(* Logix 5000 project; controller Test Emulate 5570 rev 32.11; software revision 32.00 *)

TASK MainTask (continuous, watchdog 500 ms) : MainProgram

MODULES
   Local : Emulate 5570 (ICP 5, rev 32.11)
END_MODULES

TYPE Jeyc_data :
STRUCT
   a : BOOL;
   b : BOOL;
   c : BOOL;
END_STRUCT
END_TYPE

TYPE TestUDT :
STRUCT
   b : BOOL;
END_STRUCT
END_TYPE

VAR_GLOBAL   (* controller tags *)
   HOLD : BOOL; {access Read Only}
   PROG1 : BOOL; {access Read Only}
   PROG2 : BOOL; {access Read Only}
   Reset : BOOL; {access Read Only}
   RESUME : BOOL; {access Read Only}
   SPEED : SINT; {access Read Only}
   Start : BOOL; {access Read Only}
   Stop : BOOL; {access Read Only}
END_VAR

PROGRAM MainProgram   (* main routine MainRoutine *)
VAR
   dest : SINT := 13;
   ini : SINT := 93;
   msk : SINT := 15;
   n_dest : Jeyc_data;
   n_msk : Jeyc_data := (b := 1);
   n_src : Jeyc_data := (b := 1, c := 1);
   Start : BOOL;
   Start_LT : BOOL;
   test_UDT : TestUDT; {access Read Only}
END_VAR

ROUTINE MainRoutine   (* ladder *)
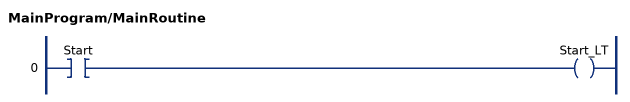
   0: XIC(Start)OTE(Start_LT);
END_ROUTINE
END_PROGRAM
